// TIA Portal V19 export
TYPE "LAF_typeConstraintWorkstationEm3ParametersInterface"
// stored: Access Published
   STRUCT
      configuration : "LAF_typeConstraintWorkstationEm3Parameters";
      commands : "LBC_typeInterfaceCommands";
      monitoring { S7_SetPoint := 'True'} : "LAF_typeConstraintWorkstationEm3ProcessValues";
   END_STRUCT;
END_TYPE
